// TIA Portal V16 export
// export: Created 2024-12-03T15:41:45.5967912Z, ExportSetting WithReadOnly, DisplayName Totally Integrated Automation Portal, DisplayVersion V16 Update 6, DisplayName TIA Portal Version Control Interface, DisplayVersion V16 Update 2, DisplayName TIA Portal Openness, DisplayVersion V16 Update 6, DisplayName TIA Portal Teamcenter Gateway, DisplayVersion V16, DisplayName SINAMICS Startdrive Advanced, DisplayVersion V16 Update 5, DisplayName SINAMICS Startdrive G130, G150, S120, S150, SINAMICS MV, S210, DisplayVersion V16 Update 5, DisplayName SINAMICS Startdrive G110M, G120, G120C, G120D, G120P, G115D, DisplayVersion V16 Update 5, DisplayName STEP 7 Professional, DisplayVersion V16 Update 6, DisplayName STEP 7 Safety, DisplayVersion V16, DisplayName WinCC Advanced / Unified PC, DisplayVersion V16 Update 6
TYPE "EVO_LABEL_STATUS_UDT"
// stored: CreationDate 2022-02-21T08:55:31.6125927Z, InterfaceModifiedDate 2022-02-21T09:23:35.2350596Z, IsConsistent true, LibraryConformanceStatus The object is library-conformant., ModifiedDate 2022-02-21T09:23:35.2350596Z
   STRUCT
      online : Bool;
      markerOk : Bool;
      applicatorOk : Bool;
   END_STRUCT;
END_TYPE
